PROGRAM MAIN
VAR
END_VAR

END_PROGRAM

(* stored: Version 1.1.0.1, ProductVersion 3.1.0.38
   POU MAIN: Id {992232b4-8414-42cf-bf25-74016d94a689}, SpecialFunc None *)
